// TwinCAT 3 PLC project PID
// ProgramVersion: 3.1.4023.0
// libraries:
//   Tc2_Standard, * (Beckhoff Automation GmbH)
//   Tc2_System, * (Beckhoff Automation GmbH)
//   Tc3_Module, * (Beckhoff Automation GmbH)
// project tree:
//   DUTs/ E_System_Mode.TcDUT (not stored), S_PID_Param.TcDUT, S_PT1T2_Param.TcDUT
//   / PlcTask.TcTTO
//   POUs/ FB_PID_Controller.TcPOU, FB_PT1T2_Process.TcPOU, FB_PWM.TcPOU, MAIN.TcPOU
// real-time tasks:
//   TASK PlcTask: cycle T#10ms, priority 20, ADS port 350

CONFIGURATION PID
    RESOURCE PLC ON TwinCAT3
        TASK PlcTask(INTERVAL := T#10ms, PRIORITY := 20);
        PROGRAM MAIN WITH PlcTask : MAIN;
    END_RESOURCE
END_CONFIGURATION

// ---- DUTs/S_PID_Param.TcDUT
TYPE S_PID_Param :
STRUCT
	Kp		: REAL;		// Reglerverstaerkung
	Ti		: REAL;		// I Anteil
	Td 		: REAL; 	// D Anteil
	N		: UINT;		// D-Anteil Filterung
	Tr		: REAL;		// Weight of Anti reset windup back calculation
	ARW		: BOOL;		// Anti reset Windup aktiv
	umin	: REAL;		// Steuergroesse minimaler Wert
	umax	: REAL;		// Steuergroesse maximaler Wert
END_STRUCT
END_TYPE

// ---- DUTs/S_PT1T2_Param.TcDUT
TYPE S_PT1T2_Param :
STRUCT
	K		: REAL;
	T1		: REAL;
	T2		: REAL;
END_STRUCT
END_TYPE

// ---- POUs/MAIN.TcPOU
PROGRAM MAIN
VAR
	PT1T2_Param		: S_PT1T2_Param;	// Parameter des Prozess
	PID_Param		: S_PID_Param;		// Parameter des Reglers
	Mode			: E_System_Mode := E_System_Mode.System_Init;	// Aktueller Modus
	T				: REAL;				// Abtastzeit
	t_run			: REAL;				// Aktuelle Laufzeit
	PID_1			: FB_PID_Controller;// PID Regler Instanz
	PT1T2_1			: FB_PT1T2_Process; // PT1T2 System Instanz
	PWM_1			: FB_PWM;			// PWM generator
	ref				: REAL;				// Referenzgroesse
	y_k				: REAL;				// Aktuelle Regelgroesse
	u_k				: REAL;				// Aktuelle Steuergroesse
END_VAR

VAR CONSTANT
	f_pwm				: REAL := 10;		// PWM Frequency
	w_pwm				: REAL := 2*PI*f_pwm;	// PWM radi
END_VAR

CASE Mode OF
	E_System_Mode.System_Init:
		// initialize variables
		ref := 0;
		y_k := 0;
		u_k := 0;
		T := 0.001;
	
		// set process variables
		PT1T2_Param.K 	:= 10;
		PT1T2_Param.T1 	:= 0.1;
		PT1T2_Param.T2 	:= 0.01;
		
		PID_Param.Kp 	:= 1/PT1T2_Param.K;
		PID_Param.Ti 	:= PT1T2_Param.T1;
		PID_Param.Td	:= PT1T2_Param.T2;
		PID_Param.Tr	:= (PID_Param.Td+PID_Param.Ti)/2;
		PID_Param.N	 	:= 10;
		PID_Param.umin  := 0;
		PID_Param.umax	:= 10;
		PID_Param.ARW 	:= TRUE;
		

		
		// call process and controller to initialize them
		PT1T2_1(u := 0, Mode := Mode, Param := PT1T2_Param, T := T);
		PID_1(ref := 0, y := 0, Mode := Mode, Param := PID_Param, T := T);
		
		// change to run mode
		Mode := E_System_Mode.System_Run;
		
	E_System_Mode.System_Run:
		// increment time
		t_run := t_run + T;
		
		// PWM Signal generator
		PWM_1(dutyPct := 50, ymin := 25, ymax := 1000, w := w_pwm, t := t_run);
		//ref := PWM_1.y;

		// call controller
		PID_1(ref := ref, y := y_k, Mode := Mode, Param := PID_Param, T := T);
		u_k := PID_1.u_sat;
		
		// call process
		PT1T2_1(u := u_k, Mode := Mode, Param := PT1T2_Param, T := T);
		y_k := PT1T2_1.y;
		
	ELSE  // default assignment
	;
		
END_CASE

END_PROGRAM

// ---- POUs/FB_PID_Controller.TcPOU
FUNCTION_BLOCK FB_PID_Controller
VAR_INPUT
	ref		: REAL;		// Aktuelle Referenzgroesse (Soll-Groesse)
	y		: REAL;		// Aktuelle Regelgroesse (Ist-Groesse)
	Mode	: E_System_Mode; 	// Aktueller Modus
	Param	: S_PID_Param;		// PID Regler Parameter
	T		: REAL;				// Abtastzeit
END_VAR
VAR_OUTPUT
	u_k		: REAL; 			// Ausgangsgroesse
	u_sat	: REAL; 			// Ausgangsgroesse gesaettigt
END_VAR
VAR
	e_k 	: REAL;
	e_k_1	: REAL;
	u_p		: REAL;
	u_i		: REAL;
	u_d		: REAL;
	u_i_k_1	: REAL;
	u_aw	: REAL;				// anti reset windup back calculation result
	bi		: REAL;				// calculation parameter for I term
	bd		: REAL;				// calculation parameter for D term
	ad		: REAL;				// calculation parameter for D term
	
END_VAR

CASE Mode OF
	E_System_Mode.System_Init:
		// calculate coefficients
		bi := Param.Kp/Param.Ti;
		ad := Param.Td / (Param.Td + Param.N * T);
		bd := (Param.Kp * Param.N * Param.Td) / (Param.Td + Param.N * T);
		
		// reset values
		//u_i_k_1	:= 0;
		//e_k_1	:= 0;
		u_aw	:= 0;
		
	E_System_Mode.System_Run:
		// implements differencial equation
		
		// compute the error
		e_k := ref - y;
		
		// proportinal term
		u_p := Param.Kp * e_k;
		
		// integral term (Trapezregel)
		u_i := u_i_k_1 + bi * (e_k + e_k_1) / 2.0 * T;
		IF Param.ARW THEN
			u_i := u_i + u_aw;
		END_IF
		
		// derivative term with filter
		u_d	:= ad * u_d + bd * (e_k - e_k_1);
		
		// total command
		u_k := u_p + u_i + u_d;
		
		// saturation
		u_sat := u_k;
		IF u_k > Param.umax THEN
			u_sat := Param.umax;
		ELSIF u_k < Param.umin THEN
			u_sat := Param.umin;
		END_IF
		
		// anti reset windup
		IF Param.ARW THEN
			u_aw := (T/Param.Tr) * (u_sat - u_k);
		END_IF
		
		// store vars for next step
		u_i_k_1 := u_i; 
		e_k_1 := e_k;
		
	ELSE  // default assignment
	;
		
END_CASE

END_FUNCTION_BLOCK

// ---- POUs/FB_PT1T2_Process.TcPOU
FUNCTION_BLOCK FB_PT1T2_Process
VAR_INPUT
	u		: REAL;				// Aktuelle Steuergroesse
	Mode	: E_System_Mode;	// Aktueller Modus
	Param	: S_PT1T2_Param;	// Parameter vom PT1T2 Modell
	T		: REAL;				// Abtastzeit
END_VAR
VAR_OUTPUT
	y 		: REAL;				// Ausgangsgroesse
END_VAR
VAR
	a1		: REAL;
	a2		: REAL;
	b0 		: REAL;
	b1		: REAL;
	c1		: REAL;
	c2		: REAL;
	y_k_1	: REAL;
	y_k_2	: REAL;
	u_k_1	: REAL;
	u_k_2	: REAL;
END_VAR

CASE Mode OF
	E_System_Mode.System_Init:
		// calculate coefficients
		a1 := EXP(-T/Param.T1);
		a2 := EXP(-T/Param.T2);
		b0 := (Param.K/(Param.T1-Param.T2))*(Param.T1*(1-a1)-Param.T2*(1-a2));
		b1 := (Param.K/(Param.T1-Param.T2))*(Param.T2*a1*(1-a2)-Param.T1*a2*(1-a1));;
		c1 := -(a1 + a2);
		c2 := a1 * a2;
		
	E_System_Mode.System_Run:
		// implements differencial equation
		y := b0*u_k_1 + b1*u_k_2 - c1*y_k_1 - c2*y_k_2;
		
		// store vars
		u_k_2 := u_k_1;
		u_k_1 := u;
		y_k_2 := y_k_1;
		y_k_1 := y;
		
	ELSE  // default assignment
	;
		
END_CASE

END_FUNCTION_BLOCK

// ---- POUs/FB_PWM.TcPOU
FUNCTION_BLOCK FB_PWM
VAR_INPUT
	dutyPct	: REAL;	// Duty cycle (%)
	ymin	: REAL; // Minimalwert
	ymax	: REAL;	// Maximalwert
	w		: REAL; // Kreisfrequenz (rad/s)
	t		: REAL; // Time (s)
END_VAR
VAR_OUTPUT
	y		: REAL; // pwm signal
END_VAR
VAR
	t_elapsed: REAL := 0;  // time since start of pwm cycle [s]
	last_t	: REAL := 0; // time since last call	
	t_cycle	: REAL; // T [s]
	t_duty	: REAL; // time when the duty cycle is over
END_VAR

// add up elapsed time
t_elapsed := t_elapsed + (t - last_t);
last_t := t;

// calc times
t_cycle := (2.0 * 3.14) / w;
t_duty := (dutyPct / 100.0) * t_cycle;

// set new t_start (either when the cylce time is reached or when t_elapsed is negative (failsafe))
IF(t_elapsed > t_cycle OR t_elapsed < 0) THEN
	t_elapsed := 0;
END_IF

// set pwm signal value
IF (t_elapsed > t_duty) THEN
	y := ymin;
ELSE
	y := ymax;
END_IF

END_FUNCTION_BLOCK
